{attribute 'linkalways'} 
{attribute 'no_explicit_call' := 'This FB is a CLASS and must be accessed using methods or properties'}
{attribute 'enable_dynamic_creation'}
FUNCTION_BLOCK _STRING EXTENDS DatatypeBase
VAR
	localData : T_MaxString;
	activeData : REFERENCE TO T_MaxString REF= localData;
END_VAR

PROPERTY PUBLIC Address : PVOID
GET
Address := ADR(activeData);
END_GET
END_PROPERTY

METHOD PUBLIC ClearReference
VAR_INPUT
END_VAR
activeData REF= localData;
END_METHOD

METHOD PUBLIC Clone : I_Datatype
VAR
    pClone : POINTER TO _STRING;
END_VAR
pClone := __NEW(_STRING(InitialValue := Value));
Clone := pClone^;
END_METHOD

METHOD FB_init : BOOL
VAR_INPUT
	bInitRetains : BOOL; // if TRUE, the retain variables are initialized (warm start / cold start)
	bInCopyCode : BOOL;  // if TRUE, the instance afterwards gets moved WORDo the copy code (online change)
	InitialValue : T_MaxString;
END_VAR
localData := InitialValue;
END_METHOD

PROPERTY PUBLIC IecType : T_MAXSTRING
GET
IecType := 'STRING';
END_GET
END_PROPERTY

METHOD PUBLIC MakeReferenceTo
VAR_INPUT
	ReferenceTarget : REFERENCE TO T_MaxString;
END_VAR
activeData REF= ReferenceTarget;
END_METHOD

METHOD PUBLIC SerializeWith
VAR_INPUT
	Serializer : I_Serializer;
END_VAR
Serializer.AddString(activeData);
END_METHOD

PROPERTY PUBLIC Size : UDINT
GET
Size := SIZEOF(activeData);
END_GET
END_PROPERTY

METHOD TryDeserializeFrom : BOOL
VAR_INPUT
	Deserializer : I_Deserializer;
	Feedback : I_DeserializerFeedback;
END_VAR
TryDeserializeFrom := Deserializer.TryGetString(activeData, Feedback);
END_METHOD

METHOD TryMakeReferenceTo : BOOL
VAR_INPUT
	Target : I_Datatype;
END_VAR
VAR
	pTargetData : POINTER TO T_MaxString;
END_VAR
IF NOT (Target.IecType = IecType) THEN
	RETURN;
END_IF

pTargetData := Target.Address;
activeData REF= pTargetData^;
TryMakeReferenceTo := TRUE;
END_METHOD

PROPERTY PUBLIC Value : T_MaxString
GET
Value := activeData;
END_GET
SET
activeData := Value;
END_SET
END_PROPERTY

END_FUNCTION_BLOCK

(* stored: Version 1.1.0.1, ProductVersion 3.1.4024.12
   POU _STRING: Id {adeac28d-1c03-0f1a-352e-189216d98317}, SpecialFunc None
   Folder Constructor: Id {28d2c79d-7aee-08ab-20c5-0859da39b9e3}
   Property Address: Id {114840a4-12ec-0738-233d-77cbf3a92971}
   Get Get: Id {87fa8174-7e1e-0b12-2ef1-8aa56d00285d}
   Method ClearReference: Id {7e45aa50-a1b6-0477-256b-58aa56ad641d}
   Method Clone: Id {124a06db-ba0c-0efe-2945-7cb763d6e2a1}
   Method FB_init: Id {389437c0-6b47-0fc4-022d-e5a2725e77e5}
   Property IecType: Id {44e03fa7-ffdb-0b18-2db4-770fb385b000}
   Get Get: Id {0309e4a8-2c3d-0d8c-0af8-8ec954adc0dd}
   Method MakeReferenceTo: Id {170da9f2-3cff-0b43-189a-ab0bcd37d445}
   Method SerializeWith: Id {a3f6077c-8b71-0b42-2f92-d07e7de399f3}
   Property Size: Id {f986a1f5-2b4a-0823-3fe9-f1e4caa82d01}
   Get Get: Id {d7817caf-635a-0e27-3c07-04b16d564dac}
   Method TryDeserializeFrom: Id {c77e8977-e056-0ec5-3869-646b3fa7298e}
   Method TryMakeReferenceTo: Id {bf372916-67cd-0817-0a6f-95bc847f2fb5}
   Property Value: Id {c07764ba-91e4-00f0-3ba1-7cfbd679b60a}
   Get Get: Id {ed26602e-a9fb-0de2-14a1-5a8b1a3c15df}
   Set Set: Id {79d655d4-9128-062e-0b35-4b082c85f51a} *)
